(* IEC 61131-3 sources: CS_4_Aufzugsteuerung/src/Stations/CP112/Steuerung/Class/clsTuerantrieb, 1 file *)

(* ---- clsTuerantrieb.st ---- *)
(*!
<Class
	Name               = "clsTuerantrieb"
	Revision           = "0.0"
	RealtimeTask       = "false"
	CyclicTask         = "true"
	DefCyclictime      = "1 ms"
	BackgroundTask     = "false"
	Sigmatek           = "false"
	OSInterface        = "false"
	HighPriority       = "false"
	Automatic          = "false"
	UpdateMode         = "Prescan"
	SharedCommandTable = "true"
	Objectsize         = "(284,120)">
	<Channels>
		<Server Name="ClassSvr" Visualized="false" Initialize="false" WriteProtected="true" Retentive="false"/>
		<Client Name="cFahrbefehl" Required="false" Internal="false"/>
	</Channels>
</Class>
*)
clsTuerantrieb : CLASS
  //Servers:
	ClassSvr 	: SvrChCmd_DINT;
  //Clients:
	cFahrbefehl 	: CltChCmd_clsMotorControl;
  //Variables:
		iStep 	: DINT;
  //Functions:

	FUNCTION VIRTUAL GLOBAL CyWork
		VAR_INPUT
			EAX 	: UDINT;
		END_VAR
		VAR_OUTPUT
			state (EAX) 	: UDINT;
		END_VAR;

	FUNCTION GLOBAL Fahrt
		VAR_INPUT
			xDir 	: BOOL;
			xStart 	: BOOL;
		END_VAR
		VAR_OUTPUT
			xBusy 	: BOOL;
		END_VAR;
  //Tables:
	FUNCTION @STD
		VAR_OUTPUT
			ret_code	: CONFSTATES;
		END_VAR;
	FUNCTION GLOBAL TAB @CT_;
END_CLASS;

#pragma usingLtd clsMotorControl

FUNCTION VIRTUAL GLOBAL  clsTuerantrieb::CyWork
VAR_INPUT
    EAX : UDINT;
END_VAR
VAR_OUTPUT
    state (EAX) : UDINT;
END_VAR

CASE iStep OF

    0: // Stillstand
        cFahrbefehl.stopNORMAL();

    10: // PowerOn positiv
        cFahrbefehl.powerOn();

        IF cFahrbefehl.sMode = clsMotorControl::MOTOR_MODE::POWER_ON THEN
            iStep := 20;
        END_IF;

    20: // Fahren positiv
        cFahrbefehl.moveABS(position:=1215752192, velocity:=800000, acceleration:=1215752192);

    30: // PowerOn negativ
        cFahrbefehl.powerOn();

        IF cFahrbefehl.sMode = clsMotorControl::MOTOR_MODE::POWER_ON THEN
            iStep := 40;
        END_IF;

    40: // Fahren negativ
        cFahrbefehl.moveABS(position:=-1215752192, velocity:=800000, acceleration:=1215752192);

    99: // Stop
        cFahrbefehl.stopNORMAL();
        iStep := 0;

ELSE
    iStep := 99;

END_CASE;

state := READY;

END_FUNCTION

FUNCTION GLOBAL clsTuerantrieb::Fahrt
VAR_INPUT
    xDir   : BOOL; // TRUE = hoch/positiv, FALSE = runter/negativ
    xStart : BOOL;
END_VAR
VAR_OUTPUT
    xBusy  : BOOL;
END_VAR

IF xStart THEN

    IF xDir THEN
        IF (iStep <> 10) AND (iStep <> 20) THEN
            iStep := 10;
        END_IF;
    ELSE
        IF (iStep <> 30) AND (iStep <> 40) THEN
            iStep := 30;
        END_IF;
    END_IF;

    xBusy := TRUE;

ELSE

    IF iStep <> 0 THEN
        iStep := 99;
    END_IF;

    xBusy := FALSE;

END_IF;

END_FUNCTION
